TYPE ST_ItemPK2_OUT2 :
STRUCT
	Identity		:ST_Identity_PK2_OUT2;
	ItemState		:STRING;
	RejectReason	:ST_RejectReason_PK2_OUT2;
	logs			:ST_logs_PK2_OUT2;
	NoRead			:STRING;
END_STRUCT
END_TYPE

(* stored: Version 1.1.0.1, ProductVersion 3.1.4024.13
   DUT ST_ItemPK2_OUT2: Id {949ce963-7f1e-4c00-9e0a-87f70d2d4b08} *)
